(* CODESYS project e!C_Visu_Test_1.ECP

Project tree, tasks and I/O mapping:
  PFC200_CS_2ETH_RS_CAN_DPS : 750-8206 PFC200 2ETH RS CAN DPS, WAGO, order no. 0750-8206, version 5.11.1.16
    application Application
      libraries: ; VisuDialogs, * (System)
      task PLC_Task (cyclic, interval t#10ms, priority 14) calls PLC_PRG
      task VISU_TASK (cyclic, interval 100 ms, priority 15) calls VisuElems.Visu_Prg
      program PLC_PRG [ST]
      visualisation Visu_A
      visualisation Visu_B
      visualisation Visu_C
    DeviceAdapter
    Kbus : Kbus, WAGO, version 1.4.0.2
        unmapped channels: K-BUS diagnostics
      _8_DO_DI_Generic : 075x-8DO8DI, WAGO, order no. 075x-8DO8DI, version 0.0.0.13
          settings: K-BUS Module slot index = 1
          unmapped channels: _IN, _OUT
        DeviceAdapter
      _4_AO_0_10V_DC : 0750-0559, WAGO, order no. 0750-0559, version 0.0.0.13
          settings: K-BUS Module slot index = 2
          unmapped channels: _QW 1, _QW 2, _QW 3, _QW 4
        DeviceAdapter
      _4_AI_10V_DC_s_e : 0750-0457, WAGO, order no. 0750-0457, version 0.0.0.9
          settings: K-BUS Module slot index = 3
          unmapped channels: _IW 1, _IW 2, _IW 3, _IW 4
        DeviceAdapter
      RS_232_RS_485_Interface_adjustable : 0750-0652, WAGO, order no. 0750-0652, version 0.0.0.25
          settings: K-BUS Module slot index = 4
          unmapped channels: _INPUTCHANNEL, _OUTPUTCHANNEL
        DeviceAdapter
    MODBUS
      MODBUS : MODBUS, WAGO, order no. n/a, version 1.1.1.15
    PROFIBUS
      PROFIBUS : PROFIBUS, WAGO, version 1.0.0.0 (disabled)
    CANbus
    Serial
      COM1 : COM1, WAGO, version 0.0.0.19
  libraries: WagoVisuIcons, 1.0.0.8 (WAGO)
  text list GlobalTextList
*)

// PFC200_CS_2ETH_RS_CAN_DPS/Application/PLC_PRG
PROGRAM PLC_PRG
VAR
	TON_SineSample: TON;
	tSineSample: TIME := T#100ms;
	rAngel: REAL;
	rSine: REAL;
	(*sWebUrl: STRING := 'http://192.168.1.32/plc/webvisu.htm';*)	
	(*sWebUrl: STRING := 'http://cam.linpro.no/view/viewer_index.shtml?id=269590';*)
	sWebUrl: STRING := 'https://video.nest.com/embedded/live/IP9Tun?autoplay=1';
	xWebShowUrl: BOOL;
	xWebBack: BOOL;
	xWebForward: BOOL;
END_VAR



TON_SineSample(IN:= TRUE, PT:= tSineSample);
IF (TON_SineSample.Q = TRUE) THEN
	TON_SineSample(IN:= FALSE);
	rAngel := rAngel + 0.1;
	rSine := 100*SIN(rAngel);  
END_IF

xWebShowUrl;
xWebBack;
xWebForward;
sWebUrl;

END_PROGRAM

// PFC200_CS_2ETH_RS_CAN_DPS/Application/Visu_A
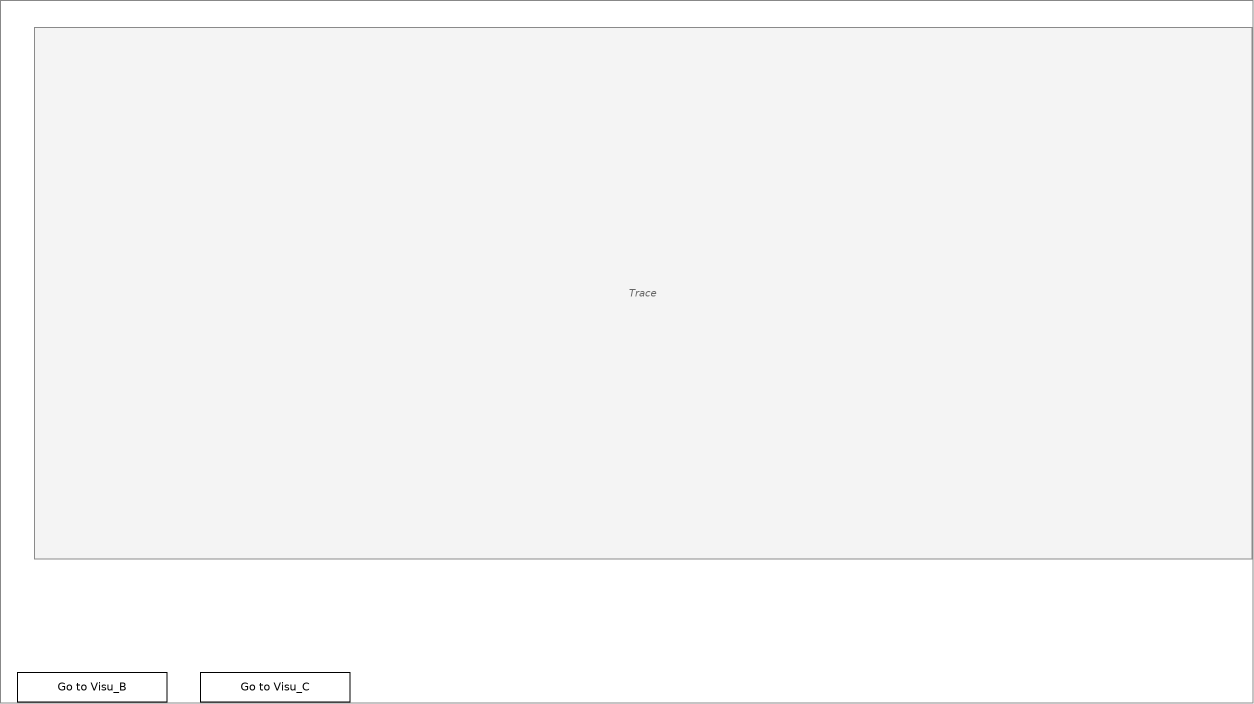
VISUALIZATION Visu_A  // 1254x704
    Trace (34,27 1218x532)
    RoundedRectangle (17,672 150x30), "Go to Visu_B"
        OnMouseDown:  Assign=Visu_B, Type=Assignment
    RoundedRectangle (200,672 150x30), "Go to Visu_C"
        OnMouseDown:  Assign=Visu_C, Type=Assignment
END_VISUALIZATION

// PFC200_CS_2ETH_RS_CAN_DPS/Application/Visu_B
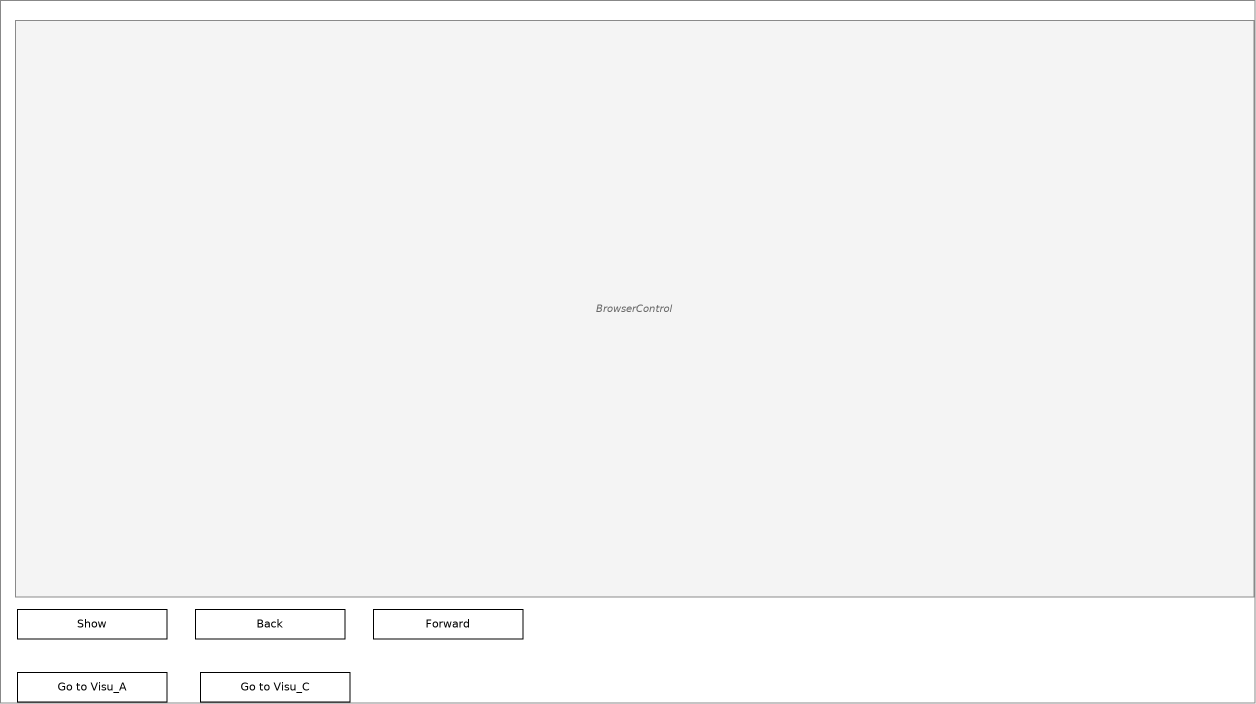
VISUALIZATION Visu_B  // 1256x704
    RoundedRectangle (17,672 150x30), "Go to Visu_A"
        OnMouseDown:  Assign=Visu_A, Type=Assignment
    BrowserControl (15,20 1239x577)
        p3734058945: PLC_PRG.sWebUrl
        p2179181546: PLC_PRG.xWebShowUrl
        p2928617338: PLC_PRG.xWebBack
        p728663958: PLC_PRG.xWebForward
    RoundedRectangle (195,609 150x30), "Back"
        tap PLC_PRG.xWebBack
    RoundedRectangle (373,609 150x30), "Forward"
        tap PLC_PRG.xWebForward
    RoundedRectangle (17,609 150x30), "Show"
        OnMouseDown: execute { PLC_PRG.xWebShowUrl := TRUE; }
    RoundedRectangle (200,672 150x30), "Go to Visu_C"
        OnMouseDown:  Assign=Visu_C, Type=Assignment
END_VISUALIZATION

// PFC200_CS_2ETH_RS_CAN_DPS/Application/Visu_C
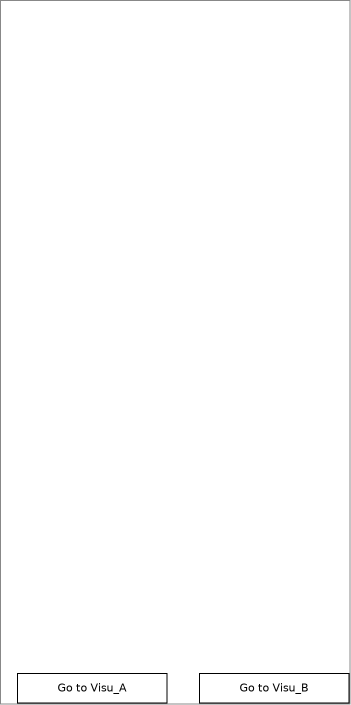
VISUALIZATION Visu_C  // 351x705
    RoundedRectangle (17,673 150x30), "Go to Visu_A"
        OnMouseDown:  Assign=Visu_A, Type=Assignment
    RoundedRectangle (199,673 150x30), "Go to Visu_B"
        OnMouseDown:  Assign=Visu_B, Type=Assignment
END_VISUALIZATION
